Universal Robots PolyScope program: g_str.urp

Program g_str (installation=ext_control directory=/programs createdIn=5.17.3 lastSavedIn=5.17.3 robotSerialNumber=20245501435)
Calibrated DH parameters: a=[0.000154, -0.137004, -0.385524, -0.00002, 0.000092, 0]; d=[0.162441, 211.794786, -230.585024, 18.923638, 0.099786, 0.09951]; alpha=[1.569493, -0.001902, 0.003874, 1.570111, -1.570167, 0]; deltaTheta=[0, -1.242934, 1.056292, 0.186646, 0.000002, 0.000001]
InitVariablesNode
Robot Program (runOnlyOnce=false)
  MoveL speed 250 mm/s, acceleration 1200 mm/s^2 (useActiveTCP=true) feature=Base
    Waypoint Waypoint_1: TCP in base x=244.537 y=603.172 z=91.747 mm, rx=-1.7467 ry=-2.0948 rz=0.8077 rad; joints [-130.747, -35.867, 89.817, -110.043, -73.974, -145.761] deg; TCP offset x=28.21 y=-96.107 z=-99.69 mm, rx=0 ry=0 rz=0 rad
    Waypoint Waypoint_2 (Relative): relativeFromPosition TCP in base x=244.521 y=603.182 z=91.749 mm, rx=-1.7467 ry=-2.0948 rz=0.8077 rad; joints [-130.745, -35.867, 89.817, -110.044, -73.975, -145.76] deg; TCP in base x=300.327 y=207.838 z=8.82 mm, rx=-1.2367 ry=-1.7305 rz=1.136 rad; joints [-170.03, -34.371, 126.934, -113.556, -94.765, -185.278] deg
